// TIA Portal V17 export
// export: Created 2022-04-06T07:28:40.8577334Z, ExportSetting WithDefaults, DisplayName Totally Integrated Automation Portal, DisplayVersion V17, DisplayName TIA Portal Openness, DisplayVersion V17, DisplayName TIA Portal Version Control Interface, DisplayVersion V17, DisplayName TIA Portal Test Suite Advanced, DisplayVersion V17, DisplayName SINAMICS Startdrive Advanced, DisplayVersion V17, DisplayName SINAMICS Startdrive G130, G150, S120, S150, SINAMICS MV, S210, DisplayVersion V17, DisplayName SINAMICS Startdrive G110M, G120, G120C, G120D, G120P, G115D, DisplayVersion V17, DisplayName STEP 7 Professional, DisplayVersion V17, DisplayName STEP 7 Safety, DisplayVersion V17, DisplayName WinCC Advanced / Unified PC, DisplayVersion V17
TYPE "LAxisCtrl_typeAxisConfig"
TITLE = LAxisCtrl_typeAxisConfig
// Support: tech.team.motioncontrol@siemens.com
// stored: IsFailsafeCompliant false
   STRUCT
      generalSettings : "LAxisCtrl_typeGeneralSettings";   // Configuration of general settings
      power : "LAxisCtrl_typePower";   // Configuration of MC_POWER function
      jog : "LAxisCtrl_typeJog";   // Configuration of JOG function
      moveVelocity : "LAxisCtrl_typeMoveVelocity";   // Configuration of MC_MOVEVELOCITY function
      stop : "LAxisCtrl_typeStop";   // Configuration of MC_HALT function
      fastStop : "LAxisCtrl_typeFastStop";   // Configuration of MC_HALT function (alternative dynamics)
      torqueLimiting : "LAxisCtrl_typeTorqueLimiting";   // Configuration of MC_TORQUELIMITING function
      homing : "LAxisCtrl_typeHoming";   // Configuration of HOMING function
      posRelative : "LAxisCtrl_typePosRelative";   // Configuration of MC_MOVERELATIVE function
      posAbsolute : "LAxisCtrl_typePosAbsolute";   // Configuration of MC_MOVEABSOLUTE function
      posSuperimposed : "LAxisCtrl_typePosSuperimposed";   // Configuration of MC_MOVESUPERIMPOSED function
      gearInRelative : "LAxisCtrl_typeGearInRelative";   // Configuration of MC_GEARIN function
      gearInAbsolute : "LAxisCtrl_typeGearInAbsolute";   // Configuration of MC_GEARIN_POS function
      camIn : "LAxisCtrl_typeCamIn";   // Configuration of MC_CAMIN function
      phasing : "LAxisCtrl_typePhasing";   // Configuration of MC_PHASING function
   END_STRUCT;
END_TYPE
